// TIA Portal V17 export
// export: Created 2024-01-30T08:49:14.5749572Z, ExportSetting WithDefaults, DisplayName Totally Integrated Automation Portal, DisplayVersion V17 Update 6, DisplayName TIA Portal Openness, DisplayVersion V17 Update 6, DisplayName TIA Portal Version Control Interface, DisplayVersion V17, DisplayName STEP 7 Professional, DisplayVersion V17 Update 6, DisplayName STEP 7 Safety, DisplayVersion V17 Update 6, DisplayName WinCC Advanced, DisplayVersion V17 Update 6
FUNCTION_BLOCK "FB_Database"   // FB2, LAD
{ S7_Optimized_Access := 'TRUE' }
VERSION : 0.1
// stored: AutoNumber true, IsIECCheckEnabled false, IsRetainMemResEnabled false, MemoryReserve 100, SetENOAutomatically false, UDAEnableTagReadback false
   VAR
      task : Int;
      Task_Start : Bool;
      TON_Act_Script { S7_SetPoint := 'True'} : TON_TIME;
   END_VAR
   VAR_TEMP
      Request : Struct
         Task_001 : Bool;
         Task_002 : Bool;
         Task_003 : Bool;
         Task_004 : Bool;
      END_STRUCT;
   END_VAR
   VAR CONSTANT
      S001_Get_Data : Int := 1;
      S002_Write_Data : Int := 2;
   END_VAR
BEGIN

NETWORK
TITLE = Reset Task Requests
// Reset Task Requests
      A     "GDB_HMI".Database.Reset_Task;
      R     "GDB_Database".Requests.Read_from_DB;
      R     "GDB_Database".Requests.Write_to_DB;



REGION Network 2 (SCL): Task Start Request
   #Request.Task_001 := "GDB_Database".Requests.Read_from_DB;
   #Request.Task_002 := "GDB_Database".Requests.Write_to_DB;
END_REGION

REGION Network 3 (SCL): 10 = Request for read Global Data
   // Set task
   IF #Request.Task_001 AND (#task = 0) THEN
       #task := 10;
   END_IF;


   //Fullfill task
   IF #task = 10 THEN

       // If reading is done
       IF "GDB_Database".Communication.Done = #S001_Get_Data AND NOT "GDB_Database".Task_Done.Read_from_DB AND "GDB_Database".Communication.Error = 0 THEN

           // Write Data from DB Receive ( on HMI Tags ) to DB on SPS
          // "GDB_HMI".Received_Data_from_DB.Rob_PRG := "GDB_Database".Receive.Rob_PRG;
          // "GDB_HMI".Received_Data_from_DB.Force := "GDB_Database".Receive.Force;
           // Set that Task is active
           "GDB_Database".Task_Done.Read_from_DB := TRUE;

       END_IF;

       // Control script
       IF #Request.Task_001 THEN
           "GDB_Database".Communication.Function := #S001_Get_Data;
           #Task_Start := TRUE;
       ELSE
           "GDB_Database".Communication.Function := 0;
           #Task_Start := FALSE;
           IF NOT "GDB_Database".Communication.Active AND "GDB_Database".Communication.Done = 0 THEN
               #task := 0;
           END_IF;
       END_IF;
   END_IF;

   // Reset Done
   IF NOT #Request.Task_001 THEN
       "GDB_Database".Task_Done.Read_from_DB := FALSE;
   END_IF;
END_REGION

REGION Network 4
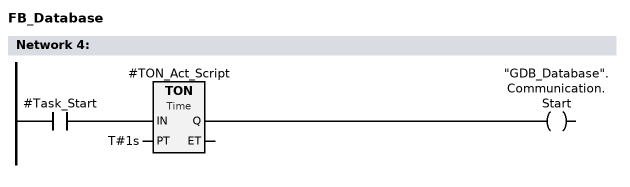
   RUNG wire#powerrail
      Contact( #Task_Start )
      { S7_Templates := "time_type := Time" } #TON_Act_Script.TON(pt := T#1s, et =>)
      Coil( "GDB_Database".Communication.Start )
   END_RUNG
   // the same network as SCL:
   #TON_Act_Script(IN := #Task_Start, PT := T#1s);   // TON
   "GDB_Database".Communication.Start := #TON_Act_Script.Q;
END_REGION
END_FUNCTION_BLOCK
